FUNCTION_BLOCK BasicPID (* Basic Function Block Type *)
  (* Standard: 61499-2 *)
  (* Version 0.0, 2011-12-09, 4DIAC-IDE, 4DIAC-Consortium *)
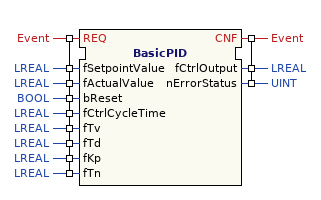
  EVENT_INPUT
    REQ WITH fSetpointValue, fActualValue, bReset, fCtrlCycleTime, fTv, fTd, fKp, fTn; (* Normal Execution Request *)
  END_EVENT
  EVENT_OUTPUT
    CNF WITH fCtrlOutput, nErrorStatus; (* Execution Confirmation *)
  END_EVENT
  VAR_INPUT
    fSetpointValue : LREAL;
    fActualValue : LREAL;
    bReset : BOOL;
    fCtrlCycleTime : LREAL;
    fTv : LREAL;
    fTd : LREAL;
    fKp : LREAL;
    fTn : LREAL;
  END_VAR
  VAR_OUTPUT
    fCtrlOutput : LREAL;
    nErrorStatus : UINT;
  END_VAR
  VAR
    fE : LREAL := 0; (* Internal Variable *)
    fE_1 : LREAL := 0; (* Internal Variable *)
    fY : LREAL := 0; (* Internal Variable *)
    fY_1 : LREAL := 0; (* Internal Variable *)
    fYP : LREAL := 0; (* Internal Variable *)
    fYI : LREAL := 0; (* Internal Variable *)
    fYI_1 : LREAL := 0; (* Internal Variable *)
    fYD : LREAL := 0; (* Internal Variable *)
    fYD_1 : LREAL := 0; (* Internal Variable *)
    bInit : BOOL := 1; (* Internal Variable *)
    bIsIPart : BOOL := 0; (* Internal Variable *)
    bIsDPart : BOOL := 0; (* Internal Variable *)
    fDi : LREAL := 0; (* Internal Variable *)
    fDd : LREAL := 0; (* Internal Variable *)
    fCd : LREAL := 0; (* Internal Variable *)
    fCtrlCycleTimeOld : LREAL := 0; (* Internal Variable *)
    fKpOld : LREAL := 0; (* Internal Variable *)
    fTnOld : LREAL := 0; (* Internal Variable *)
    fTvOld : LREAL := 0; (* Internal Variable *)
    fTdOld : LREAL := 0; (* Internal Variable *)
    nERR_NOERROR : UINT := 0; (* Internal Variable *)
    nERR_INVALIDPARAM : UINT := 1; (* Internal Variable *)
    nERR_INVALIDCYCLETIME : UINT := 2; (* Internal Variable *)
  END_VAR
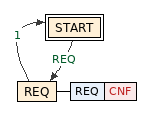
  EC_STATES
    START; (* Initial State *)
    REQ : REQ -> CNF; (* Normal execution *)
  END_STATES
  EC_TRANSITIONS
    START TO REQ := REQ;
    REQ TO START := 1;
  END_TRANSITIONS
  ALGORITHM REQ IN ST: (* Normally executed algorithm *)
(* init necessary? *)
IF (fCtrlCycleTime <> fCtrlCycleTimeOld) OR (fKp <> fKpOld) OR (fTn <> fTnOld) OR (fTv <> fTvOld) OR (fTd <> fTdOld) THEN
		bInit := TRUE;
END_IF;
(* controller init *)
IF bInit OR bReset THEN
		(* reset internal and external variables *)
		fE := fE_1 := 0.0;
		fY := fY_1 := 0.0;
		fYP := 0.0;
		fYI := fYI_1 := 0.0;
		fYD := fYD_1 := 0.0;
		fCtrlOutput := 0.0;
		bIsIPart := FALSE;
		bIsDPart := FALSE;
		fCtrlOutput := 0.0;
		nErrorStatus := nERR_NOERROR;
		(* check cycle time parameter: (CycleTime > 0 AND CycleTme <= 60) *)
		IF ( fCtrlCycleTime <= 0) THEN
			nErrorStatus := nERR_INVALIDCYCLETIME;
			RETURN;
		END_IF;
		(* check controller parameters: (Tn, Tv, Td >= 0) *)
		IF ( (fTn < 0) OR (fTv < 0) OR (fTd < 0) ) THEN
			nErrorStatus := nERR_INVALIDPARAM;
			RETURN;
		END_IF;
		(* I-part *)
		IF( fTn > 0.0 ) THEN
			fDi := (fKp * fCtrlCycleTime) / (2.0 * fTn);
			bIsIPart := TRUE;
		ELSE
			fDi := 0.0;
			bIsIPart := FALSE;
		END_IF;
		(* D-part *)
		IF( fTv > 0.0 ) AND (fTd > 0.0) THEN
			fDd := (fKp * fTv) / (fTd + fCtrlCycleTime / 2.0);
			fCd := (fTd - fCtrlCycleTime / 2.0) / (fTd + fCtrlCycleTime / 2.0);
			bIsDPart := TRUE;
		ELSE
			fDd := 0.0;
			fCd := 0.0;
			bIsDPart := FALSE;
		END_IF;
		(* reset *)
		IF bReset THEN
			RETURN;
		END_IF
		(* set internal init flag *)
		fCtrlCycleTimeOld := fCtrlCycleTime;
		fKpOld := fKp;
		fTnOld := fTn;
		fTvOld := fTv;
		fTdOld := fTd;
		bInit := FALSE;
	END_IF;
	(* 3. save old variable *)
	fE_1 := fE;
	fY_1 := fY;
	fYI_1 := fYI;
	fYD_1 := fYD;
	(* 4. set error/deviation input *)
	fE := fSetpointValue - fActualValue;
	(* 5. YP-part *)
	fYP := fKp * fE;
	(* 6. YI-part *)
	IF bIsIPart THEN
		fYI := fYI_1 + fDi * (fE + fE_1);
	 (* normal I-part calculation *)
	ELSE
		fYI := 0.0;
	END_IF;
	(* 7. YD-part *)
	IF bIsDPart THEN
		fYD := fCd * fYD_1 + fDd * (fE - fE_1);
	ELSE
		fYD := 0.0;
	END_IF;
	(* 8. Ysum = YP + YI + YD *)
	fY := fYP + fYI + fYD;
	(* 10. set controller output *)
	fCtrlOutput := fY;
  END_ALGORITHM
  SERVICE left interface/right interface (* Basic Function Block Type *)
    SEQUENCE request
      left interface.REQ() -> left interface.CNF(fCtrlOutput=[0.0,]; nErrorStatus=[0,2]);
    END_SEQUENCE
  END_SERVICE
END_FUNCTION_BLOCK
